FUNCTION_BLOCK ILOCK_SWITCH (* Prioritizes the last active input. *)
  (* Standard: 61499-2 *)
  (* Version 1.0, 2026-02-23, Franz Höpfinger *)
  PACKAGE logiBUS::signalprocessing::interlock;
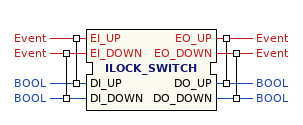
  EVENT_INPUT
    EI_UP WITH DI_UP;
    EI_DOWN WITH DI_DOWN;
  END_EVENT
  EVENT_OUTPUT
    EO_UP WITH DO_UP;
    EO_DOWN WITH DO_DOWN;
  END_EVENT
  VAR_INPUT
    DI_UP : BOOL; (* TRUE = forward, up, right, clockwise *)
    DI_DOWN : BOOL; (* TRUE = backward, down, left, counter-clockwise *)
  END_VAR
  VAR_OUTPUT
    DO_UP : BOOL; (* TRUE = forward, up, right, clockwise *)
    DO_DOWN : BOOL; (* TRUE = backward, down, left, counter-clockwise *)
  END_VAR
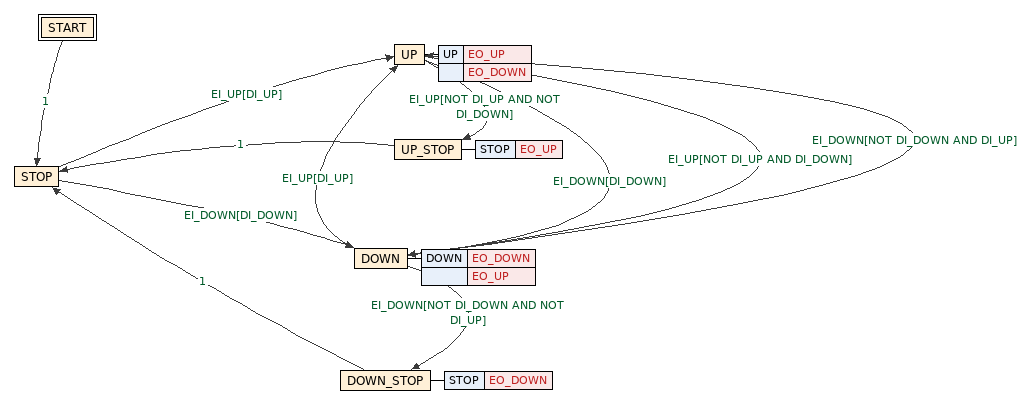
  EC_STATES
    START; (* Initial State *)
    UP : UP -> EO_UP, -> EO_DOWN;
    DOWN : DOWN -> EO_DOWN, -> EO_UP;
    STOP;
    UP_STOP : STOP -> EO_UP;
    DOWN_STOP : STOP -> EO_DOWN;
  END_STATES
  EC_TRANSITIONS
    STOP TO UP := EI_UP[DI_UP];
    STOP TO DOWN := EI_DOWN[DI_DOWN];
    UP TO DOWN := EI_DOWN[DI_DOWN];
    UP TO DOWN := EI_UP[NOT DI_UP AND DI_DOWN];
    UP TO UP_STOP := EI_UP[NOT DI_UP AND NOT DI_DOWN];
    DOWN TO UP := EI_UP[DI_UP];
    DOWN TO UP := EI_DOWN[NOT DI_DOWN AND DI_UP];
    DOWN TO DOWN_STOP := EI_DOWN[NOT DI_DOWN AND NOT DI_UP];
    UP_STOP TO STOP := 1;
    DOWN_STOP TO STOP := 1;
    START TO STOP := 1;
  END_TRANSITIONS
  ALGORITHM UP IN ST:
DO_UP := BOOL#TRUE;
DO_DOWN := BOOL#FALSE;
  END_ALGORITHM
  ALGORITHM DOWN IN ST:
DO_UP := BOOL#FALSE;
DO_DOWN := BOOL#TRUE;
  END_ALGORITHM
  ALGORITHM STOP IN ST:
DO_UP := BOOL#FALSE;
DO_DOWN := BOOL#FALSE;
  END_ALGORITHM
END_FUNCTION_BLOCK
